FUNCTION_BLOCK PAMIntake EXTENDS PAMLoadingstation
VAR_INPUT
END_VAR
VAR_OUTPUT
END_VAR
VAR
END_VAR

END_FUNCTION_BLOCK

(* stored: Version 1.1.0.1, ProductVersion 3.1.4020.12
   POU PAMIntake: Id {cac1cf61-6858-4557-b7b9-1aa9b8cdf323}, SpecialFunc None *)
